FUNCTION F_LogLA7 
VAR_INPUT
	eLogLevel		: E_LogLevel;
	sLogger			: T_MaxString;
	sMessage		: T_MaxString;
	aArg1			: ANY;
	aArg2			: ANY;
	aArg3			: ANY;
	aArg4			: ANY;
	aArg5			: ANY;
	aArg6			: ANY;
	aArg7			: ANY;
END_VAR
VAR 
	aEmptyArg		: BYTE;
END_VAR

F_LogA(
	eLogLevel,
	sLogger,
	sMessage,
	4,
	aArg1,
	aArg2,
	aArg3,
	aArg4,
	aArg5,
	aArg6,
	aArg7,
	aEmptyArg,
	aEmptyArg,
	aEmptyArg
);

END_FUNCTION

(* stored: Version 1.1.0.1, ProductVersion 3.1.4024.0
   POU F_LogLA7: Id {02326550-5720-4e83-98b1-0c77b7273581}, SpecialFunc None *)
